# EPICS substitutions: iocBoot/ioc4idVDCM/substitutions/AcsMotion_monochromator.substitutions
file "$(MOTOR)/db/asyn_motor.db"
{
pattern
{N,  M,        DTYP,         PORT,  ADDR,          DESC,    EGU,  DIR,    VELO,    VBAS,   ACCL,  BDST,   BVEL,   BACC,  MRES,             PREC,  DHLM,   DLLM,  INIT, RTSM, RTRY}
{1,  "m$(N)",  "asynMotor",  ACS1,  0,    "Bragg angle",    deg,  Pos,    0.10,    0.0001,  0.1,     0,      1,    0.2,  -5.72957795e-07,  4,     1000,  -1000,    "", "Never", 0}
{2,  "m$(N)",  "asynMotor",  ACS1,  1,              "X",     mm,  Pos,    0.10,    0.0001,  0.1,     0,      1,    0.2,  0.00005,          4,     1000,  -1000,    "", "Never", 0}
{3,  "m$(N)",  "asynMotor",  ACS1,  2,              "Y",     mm,  Pos,    0.10,    0.0001,  0.1,     0,      1,    0.2,  0.00005,          4,     1000,  -1000,    "", "Never", 0}
{4,  "m$(N)",  "asynMotor",  ACS1,  3,        "Pitch 2",    deg,  Pos,    0.08,    0.0001,  0.1,     0,      1,    0.2,  3.9184953e-6,     4,     1000,  -1000,    "", "Never", 0}
{5,  "m$(N)",  "asynMotor",  ACS1,  4,         "Roll 2",    rad,  Pos,   0.0001,  0.00001,  0.1,     0,      1,    0.2,  0.00000002677,    4,     1000,  -1000,    "", "Never", 0}
}

### The feedback database is helpful for troubleshooting encoder problems
file "$(MOTOR_ACSMOTION)/db/SPiiPlusFeedback.db"
{
pattern
{M,   PORT, ADDR, PREC, SCAN}
{m1,  ACS1,    0,    6,    2}
{m2,  ACS1,    1,    6,    2}
{m3,  ACS1,    2,    6,    2}
{m4,  ACS1,    3,    6,    2}
{m5,  ACS1,    4,    6,    2}
}

### Disable setting the position for axes with absolute encoders
file "$(MOTOR_ACSMOTION)/db/SPiiPlusDisableSetPos.db"
{
pattern
{M,   PORT, ADDR}
{m1,  ACS1,    0}
{m2,  ACS1,    1}
{m3,  ACS1,    2}
{m4,  ACS1,    3}
{m5,  ACS1,    4}
}
